# EPICS autosave request: soft_iocs/galil_DMC/iocBoot/iocgalil_DMC_E04/GalilTest_18ID_DMC_E04Positions.req
$(P)25.DVAL
$(P)26.DVAL
$(P)27.DVAL
$(P)28.DVAL
$(P)29.DVAL
$(P)30.DVAL
$(P)31.DVAL
$(P)32.DVAL
